(* PLC project Unnamed, Unknown Unnamed 1 *)
(* stored: creationDateTime 2019-04-18T11:44:44, modificationDateTime 2019-12-16T01:48:12 *)

PROGRAM controle
  VAR
    button AT %IX100.0 : BOOL;  (* BUTTON LIGA/RESET *)
    button_scada AT %QX2.0 : BOOL;  (* LIGA O CONTROLE NO SCADA *)
    lamp AT %QX100.0 : BOOL;  (* SINAL DO ERROR ZERO *)
    lamp_scada AT %QX3.0 : BOOL;  (* SINAL DO ERRO NO SCADA *)
    IN AT %IW100 : UINT;  (* SAIDA DA PLANTA RC *)
    IN_SCADA AT %QW0 : UINT;  (* SAIDA DA PLANTA RC PARA SCADA *)
    OUT AT %QW100 : INT;  (* AÇÃO DE CONTROLE *)
    OUT_SCADA AT %QW1 : INT;  (* AÇÃO DE CONTROLE PARA O SCADA *)
    SP_SCADA AT %QW2 : UINT;  (* SETPOINT DO SCADA *)
  END_VAR
  VAR
    PID0 : PID;  (* BLOCO PID *)
  END_VAR
  VAR
    KP_SCADA AT %QW3 : UINT;  (* PROPORCIONAL DO SCADA *)
    TI_SCADA AT %QW4 : UINT;  (* INTEGRAL DO SCADA *)
    TD_SCADA AT %QW5 : UINT;  (* DERIVATIVO DO SCADA *)
  END_VAR

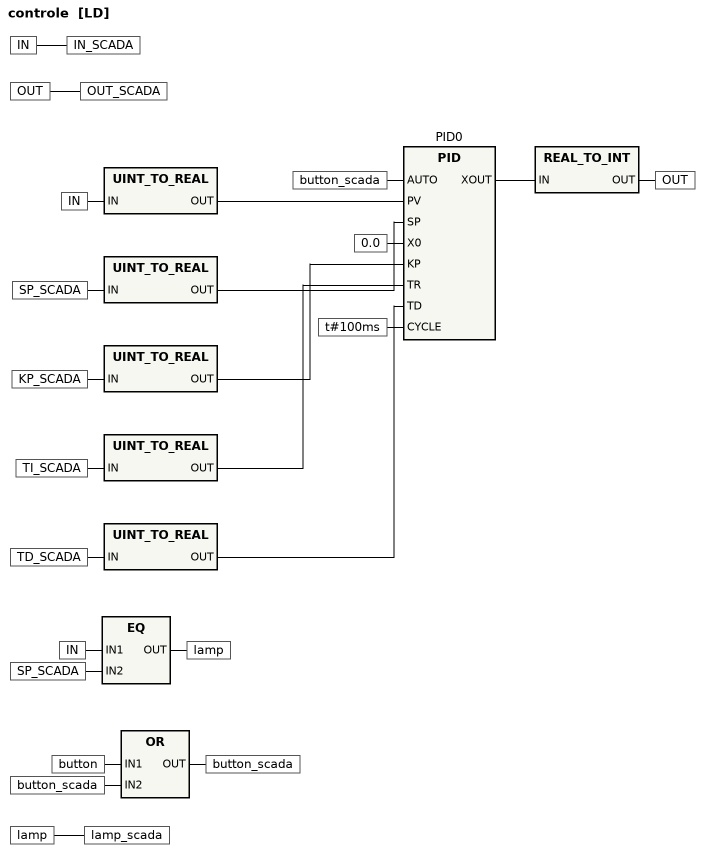
(* LD diagram, written out as Structured Text *)
IN_SCADA := IN;
PID0(AUTO := button_scada, PV := UINT_TO_REAL(IN), SP := UINT_TO_REAL(SP_SCADA), X0 := 0.0, KP := UINT_TO_REAL(KP_SCADA), TR := UINT_TO_REAL(TI_SCADA), TD := UINT_TO_REAL(TD_SCADA), CYCLE := t#100ms);
OUT := REAL_TO_INT(PID0.XOUT);
OUT_SCADA := OUT;
lamp := IN = SP_SCADA;
lamp_scada := lamp;
button_scada := button OR button_scada;
END_PROGRAM

CONFIGURATION Config0
  RESOURCE Res0 ON PLC
    TASK task0(INTERVAL := T#20ms, PRIORITY := 0);
    PROGRAM instance0 WITH task0 : controle;
  END_RESOURCE
END_CONFIGURATION
